FUNCTION_BLOCK CM_ValveWithDoubleFB EXTENDS CM_ValveWithFB
VAR_INPUT
	//Inputs (extra on top of the base valve)
	I_bStaValveIsOn2 AT %I* : BOOL; //Valve is on (on = positive logic of fuction)
	I_bStaValveIsOff2 AT %I* : BOOL; //Valve is off
	
	//Status
	s_bStaValveIsOff1 : BOOL;
	s_bStaValveIsOff2 : BOOL;
	s_bStaValveIsOn1 : BOOL;
	s_bStaValveIsOn2 : BOOL;
	
END_VAR


SUPER^();

METHOD PROTECTED _m_Alarms : BOOL
VAR_INST
	s_sTempStringOff : STRING(3);
	s_sTempStringOn : STRING(3);
END_VAR

IF NOT SUPER^._m_Alarms() THEN
	RETURN;
END_IF

// Timeout (timers)
s_tonFeedBackOffTimeout(
	IN := i_bReqEnable AND s_bReqOff AND NOT(s_bStaValveIsOff),
	PT := i_stSettings.tValveOffTimeout );
	
s_tonFeedbackOnTimeout(
	IN := i_bReqEnable AND s_bReqOn AND NOT(s_bStaValveIsOn),
	PT := i_stSettings.tValveOnTimeout );

// Set error bits
s_errFeedbackOffTimeout := (s_tonFeedBackOffTimeout.Q OR s_errFeedbackOffTimeout) AND NOT(i_bCmdReset);
s_errFeedbackOnTimeout := (s_tonFeedbackOnTimeout.Q OR s_errFeedbackOnTimeout) AND NOT(i_bCmdReset);

IF s_errFeedbackOffTimeout THEN 
	IF NOT(s_bStaValveIsOff1) AND NOT(s_bStaValveIsOff2) THEN
		s_sTempStringOff := '1&2';
	ELSIF NOT(s_bStaValveIsOff1) THEN
		s_sTempStringOff := '1';
	ELSIF NOT(s_bStaValveIsOff2) THEN
		s_sTempStringOff := '2';
	END_IF
ELSE
	s_sTempStringOff := '-';		
END_IF

IF s_errFeedbackOnTimeout THEN 
	IF NOT(s_bStaValveIsOn1) AND NOT(s_bStaValveIsOn2) THEN
		s_sTempStringOn := '1&2';
	ELSIF NOT(s_bStaValveIsOn1) THEN
		s_sTempStringOn := '1';
	ELSIF NOT(s_bStaValveIsOn2) THEN
		s_sTempStringOn := '2';
	END_IF
ELSE
	s_sTempStringOn := '-';		
END_IF

s_fbAlarmHandlerFeedbackOffTimeout(
	i_bStaActive := i_bReqEnable AND s_errFeedbackOffTimeout, 
	i_eAlarmLevel := E_AlarmLevel.Alarm,
	i_sAlarmText := CONCAT(i_sCmName, CONCAT(': Feedback off timeout - Feedback: ', s_sTempStringOff)));
	
s_fbAlarmHandlerFeedbackOnTimeout(
	i_bStaActive := i_bReqEnable AND s_errFeedbackOnTimeout, 
	i_eAlarmLevel := E_AlarmLevel.Alarm,
	i_sAlarmText := CONCAT(i_sCmName, CONCAT(': Feedback on timeout - Feedback: ', s_sTempStringOn)));

s_bStaError := 
	s_fbAlarmHandlerFeedbackOffTimeout.q_bStaActive
	OR s_fbAlarmHandlerFeedbackOnTimeout.q_bStaActive;

_m_Alarms := TRUE;
END_METHOD

METHOD PROTECTED _m_Inputs : BOOL

IF NOT SUPER^._m_Inputs() THEN
	RETURN;
END_IF

s_bStaValveIsOff1 := I_bStaValveIsOff;
s_bStaValveIsOff2 := I_bStaValveIsOff2;
s_bStaValveIsOff := s_bStaValveIsOff1 AND s_bStaValveIsOff2;

s_bStaValveIsOn1 := I_bStaValveIsOn;
s_bStaValveIsOn2 := I_bStaValveIsOn2; 
s_bStaValveIsOn := s_bStaValveIsOn1 AND s_bStaValveIsOn2;

_m_Inputs := TRUE;
END_METHOD

END_FUNCTION_BLOCK

(* stored: Version 1.1.0.1, ProductVersion 3.1.4024.12
   POU CM_ValveWithDoubleFB: Id {fa1c28a2-56d2-405b-8a48-8aed0a8180fb}, SpecialFunc None
   Method _m_Alarms: Id {325d43c3-5745-4ae0-9bdb-3517c36b11b7}
   Method _m_Inputs: Id {575f2f03-5155-4a44-a733-1df6472e24f5} *)
